{attribute 'GeneratedUsingTerminal: IODEVICETYPE_ETHERCATPROT'}
{attribute addProperty BoxType "IODEVICETYPE_ETHERCATPROT"}
{attribute addProperty Id "TcTerminals210_2EK1100TcTerminals210_2EK1100_50C143310SyncUnitsSyncUnits_99E584AF18InputsInputs_25A0042B160OutputsOutputs_2397A10E106InfoDataInfoData_C76BEFB322"}
{attribute addProperty CRC "4086334510"}
{attribute addProperty Size "306"}
TYPE EtherCAT_Master_KLxxxx_2_F390842E :
STRUCT
	{attribute addProperty Name "TcTerminals210_2EK1100"}
	{attribute addProperty PreviousPort "EtherCAT_Master_KLxxxx_2 : Master"}
	TcTerminals210_2EK1100 : TcTerminals210_2EK1100_50C14331;
	{attribute addProperty Name "SyncUnits"}
	SyncUnits : SyncUnits_99E584AF;
	{attribute addProperty Name "Inputs"}
	Inputs : Inputs_25A0042B;
	{attribute addProperty Name "Outputs"}
	Outputs : Outputs_2397A10E;
	{attribute addProperty Name "InfoData"}
	InfoData : InfoData_C76BEFB3;
END_STRUCT
END_TYPE

(* stored: Version 1.2.0.0, ProductVersion 3.1.4024.9
   DUT EtherCAT_Master_KLxxxx_2_F390842E: Id {caf9d60a-e697-4999-8a07-a8798b150597} *)
